(* PLC project model, Beckhoff Automation Beckhoff MLlib 3.1.251201.0 *)
(* stored: creationDateTime 2026-07-10T12:15:19.8299835, modificationDateTime 2026-07-10T12:15:19.8299835 *)

TYPE ST_modelInput :
STRUCT

	{attribute 'hide'} _header_DO_NOT_CHANGE : ARRAY[0..63] OF SINT := [-1,-112,120,86,52,18,-1,-1,1,-1,0,0,-1,-1,-112,-112,76,-37,-101,-100,-56,125,72,-20,-8,-106,39,-43,33,76,57,117,-100,-22,-66,-55,64,-24,-107,-56,26,-38,-68,-13,105,114,16,-98,-44,2,0,0,0,0,0,0,0,0,0,0,0,0,0,0];
	in_input_tensor : ARRAY[0..0,0..32,0..4] OF REAL;

END_STRUCT
END_TYPE

TYPE ST_modelOutput :
STRUCT

	{attribute 'hide'} _header_DO_NOT_CHANGE : ARRAY[0..63] OF SINT := [-1,-112,120,86,52,18,-1,-1,1,-1,0,0,-1,-1,-112,-112,-35,24,-50,75,-65,96,-121,123,127,87,61,127,-39,-108,16,-70,120,-89,-28,78,-43,26,-32,-7,81,19,29,-89,-55,3,43,2,68,0,0,0,0,0,0,0,0,0,0,0,0,0,0,0];
	out_prediction_tensor : ARRAY[0..0,0..0] OF REAL;

END_STRUCT
END_TYPE
